PROGRAM PRG_08_AutoCrossCut
VAR
	iStep: INT;
	TON_DownDelay: TON;
	ctu_DoublePass: CTU;
	bDoublePassCountUp: BOOL;
	TON_bAutoUp: TON;
	bTON_AutoUp: BOOL;
	R_TRIG_0: R_TRIG;
	TON_AutoCrossCutError: TON;
	SR_DoublePass: SR;
	bDoublePassQ: BOOL;
	FB_Blinker_AutoCrossCut: fb_Blinker;
	TON_AutoCrossCutWatchdog: TON;
	RS_watchdog: RS;
	R_TRIG_1: R_TRIG;
	R_TRIG_2: R_TRIG;
	R_TRIG_3: R_TRIG;
	R_TRIG_4: R_TRIG;
	R_TRIG_5: R_TRIG;
	bWatchdogReset: BOOL;
	R_TRIG_6: R_TRIG;
	R_TRIG_7: R_TRIG;
	SR_WatchdogTriggered: SR;
	bWatchdogSet: BOOL;
	iStepErr: INT;
	R_TRIG_iStepErr: R_TRIG;
END_VAR

// Watchdog timeout error step
	R_TRIG_iStepErr(CLK:= SR_WatchdogTriggered.Q1, Q=> );
	IF R_TRIG_iStepErr.Q THEN
		iStepErr := iStep;
	ELSIF IN_FaultReset AND SR_WatchdogTriggered.Q1 THEN
		iStepErr := 0;
	END_IF

	
// error
	IF		NOT bSafetyOK 
			OR IN_FaultReset 
			OR NOT OUT_bSawON 
			OR bAnyServoError 
			OR bMachineHoming 
			OR bCrossCutPosition 
			OR SR_WatchdogTriggered.Q1
			OR bRemote
	THEN	iStep	:=	0 ;
			bWatchdogReset := TRUE ;
	END_IF

(* Time delay 0.5 sec after saw blade reached the bottom limit *)	
	TON_DownDelay(IN:= , PT:= T#0.5S, Q=> , ET=> );
	IF		iStep <> 30 THEN
			TON_DownDelay.IN	:= FALSE ;
	END_IF
(* Double Pass counter BOOL *)
	IF		ctu_DoublePass.CV	=	1
	THEN	bDoublePassCountUp		:=	TRUE;
	ELSE	bDoublePassCountUp		:=	FALSE;
	END_IF

CASE iStep OF 
	0:		//	Step 0	:	Init step
				bAutoCrossCut	:= FALSE ;
				bAutoUp			:= FALSE ;
				bAutoDown		:= FALSE ;
				bAutoCut		:= FALSE ;
				bAutoReturn		:= FALSE ;
				bTON_AutoUp		:= FALSE ;
				bWatchdogReset	:= TRUE  ;
				
		IF
				bSafetyOK
				AND bTurret045Range
				AND OUT_bSawON
				AND (bAutoCrossCutEnable AND IN_bAutoCycleStart AND NOT bRemote)
				AND NOT bMachineHoming
				AND NOT bCrossCutPosition
				AND bCarriageCentreRef
		THEN
				bAutoCrossCut := TRUE	;
				bWatchdogReset := TRUE  ;
				iStep	:=		20		;
		ELSE
				bAutoCrossCut := FALSE	;
				bWatchdogReset := FALSE ;
				iStep	:=		0		;
		END_IF

	20:		// Step 20	:	Saw RETURN movement
		IF 
				bAutoCrossCut
				AND bSafetyOK
				AND NOT bCrossCutRightLimit
			
		THEN	bAutoReturn	:=	TRUE	;
				bWatchdogReset := FALSE ;
		
		ELSE
				bAutoReturn	:=	FALSE	;
				bWatchdogReset := TRUE  ;
				iStep		:=	30		;
		END_IF
	
		IF 		NOT bSafetyOK
		THEN 	
				bAutoReturn	:=	FALSE	;
				bWatchdogReset := TRUE  ;
				iStep		:=	0		;
		END_IF
		
	30:		// Step 30	:	Saw DOWN movement
	ctu_DoublePass.CV;
		IF
				bAutoCrossCut
				AND bSafetyOK
				AND ((bAutoCrossCutDoublePass AND NOT bDoublePassReference AND bDoublePassCountUp) 
					OR ( NOT SR_DownLimit.Q1 AND (bDoublePassQ OR NOT bDoublePassCountUp)))
		THEN	
				bAutoDown	:=	TRUE	;
				bWatchdogReset := FALSE ;
		ELSE
				bAutoDown	:=	FALSE	;
				TON_DownDelay.IN := TRUE ;
					IF TON_DownDelay.Q THEN
						bWatchdogReset := TRUE ;
						iStep	:=	40		;
					END_IF
		END_IF
		
		IF 		NOT bSafetyOK
		THEN 	
				bAutoDown	:=	FALSE	;
				bWatchdogReset := TRUE  ;
				iStep		:=	0		;
		END_IF
	
	40:		// Step 40	:	Saw CUT movement
		IF
				bAutoCrossCut
				AND bSafetyOK
				AND	NOT bCrossCutLeftLimit
			THEN
				bAutoCut	:=	TRUE	;
				bWatchdogReset := FALSE ;
		ELSE
				bAutoCut	:=	FALSE	;
				bWatchdogReset := TRUE	;
				iStep		:=	50		;
		END_IF
		
		IF 		NOT bSafetyOK
			THEN 	
				bAutoCut	:=	FALSE	;
				bWatchdogReset := TRUE	;
				iStep		:=	0		;
		END_IF
	
	50:		// Step 50	:	Saw UP movement		(* for double pass: only lift slightly, RETURN, then plunge all the way down *)
	ctu_DoublePass.CV;	
		IF
				bAutoCrossCutDoublePass AND bDoublePassCountUp AND NOT bDoublePassQ
			THEN
				bTON_AutoUp	:=	TRUE	;
				bWatchdogReset := FALSE ;
				bAutoUp		:=	NOT TON_bAutoUp.Q	;
				
				IF
					R_TRIG_0.Q THEN
					bWatchdogReset := TRUE ;
					iStep	:=	60	;
				END_IF
				
		ELSIF
				bAutoCrossCut
				AND bSafetyOK
				AND NOT bSawUpLimit
				AND ((bDoublePassQ AND NOT bDoublePassCountUp AND bAutoCrossCutDoublePass) OR (NOT bAutoCrossCutDoublePass))
			THEN
				bAutoUp		:=	TRUE	;
				bWatchdogReset := FALSE ;
		ELSE
				bAutoUp		:=	FALSE	;
				bWatchdogReset := TRUE	;
				iStep		:=	60		;
		END_IF
		
		IF 		NOT bSafetyOK
		THEN 	
				bAutoUp		:=	FALSE	;
				bWatchdogReset := TRUE	;
				iStep		:=	0		;
		END_IF
	
	60:		// Step 60	:	Saw RETURN movement (loop back to step 20 if double pass)
		IF
				bAutoCrossCutDoublePass
				AND bDoublePassCountUp
		THEN
				bWatchdogReset := TRUE  ;
				iStep		:=	20		;
		ELSIF	
				bAutoCrossCut
				AND bSafetyOK
				AND NOT bCrossCutCentre
		THEN
				bWatchdogReset := FALSE ;
				bAutoReturn	:=	TRUE	;
		ELSE
				bAutoReturn	:=	FALSE	;
				bWatchdogReset := TRUE	;
				iStep		:=	0		;
		END_IF
		
		IF 		NOT bSafetyOK
		THEN 	
				bAutoReturn	:=	FALSE	;
				bWatchdogReset := TRUE	;
				iStep		:=	0		;
		END_IF
END_CASE

ACTION ACT_08_1_AutoCrossCut:
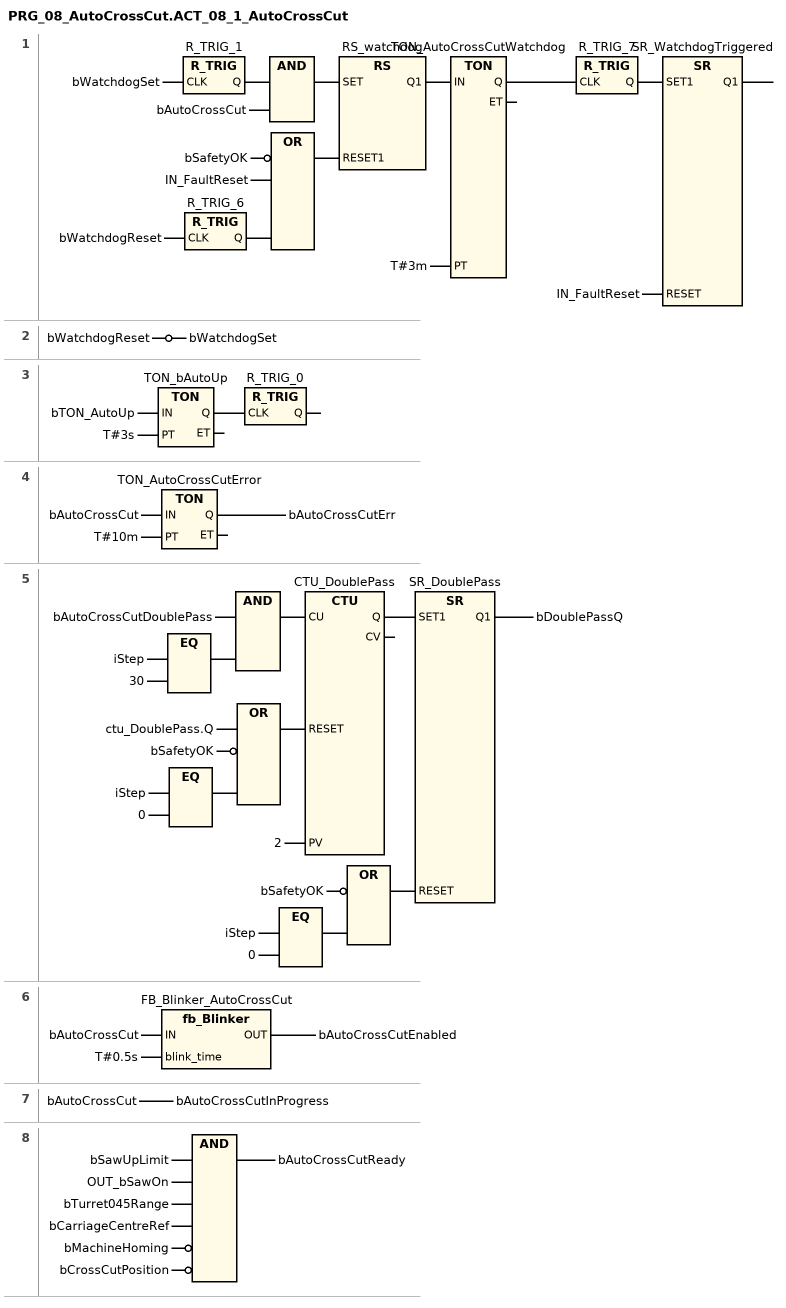
// NETWORK 1
R_TRIG_1(CLK := bWatchdogSet); // R_TRIG
R_TRIG_6(CLK := bWatchdogReset); // R_TRIG
RS_watchdog(SET := R_TRIG_1.Q AND bAutoCrossCut, RESET1 := NOT bSafetyOK OR IN_FaultReset OR R_TRIG_6.Q); // RS
TON_AutoCrossCutWatchdog(IN := RS_watchdog.Q1, PT := T#3m); // TON
R_TRIG_7(CLK := TON_AutoCrossCutWatchdog.Q); // R_TRIG
SR_WatchdogTriggered(SET1 := R_TRIG_7.Q, RESET := IN_FaultReset); // SR

// NETWORK 2
bWatchdogSet := NOT bWatchdogReset;

// NETWORK 3
TON_bAutoUp(IN := bTON_AutoUp, PT := T#3s); // TON
R_TRIG_0(CLK := TON_bAutoUp.Q); // R_TRIG

// NETWORK 4
TON_AutoCrossCutError(IN := bAutoCrossCut, PT := T#10m); // TON
bAutoCrossCutErr := TON_AutoCrossCutError.Q;

// NETWORK 5
CTU_DoublePass(
    CU := bAutoCrossCutDoublePass AND iStep = 30,
    RESET := ctu_DoublePass.Q OR NOT bSafetyOK OR iStep = 0,
    PV := 2); // CTU
SR_DoublePass(SET1 := CTU_DoublePass.Q, RESET := NOT bSafetyOK OR iStep = 0); // SR
bDoublePassQ := SR_DoublePass.Q1;

// NETWORK 6
FB_Blinker_AutoCrossCut(IN := bAutoCrossCut, blink_time := T#0.5s); // fb_Blinker
bAutoCrossCutEnabled := FB_Blinker_AutoCrossCut.OUT;

// NETWORK 7
bAutoCrossCutInProgress := bAutoCrossCut;

// NETWORK 8
bAutoCrossCutReady := bSawUpLimit AND OUT_bSawOn AND bTurret045Range AND bCarriageCentreRef AND NOT bMachineHoming AND NOT bCrossCutPosition;
END_ACTION

END_PROGRAM

(* stored: Version 1.1.0.1, ProductVersion 3.1.4024.15
   POU PRG_08_AutoCrossCut: Id {73f4070d-b53d-44b0-b7c0-d862c4fca4a8}, SpecialFunc None
   Action ACT_08_1_AutoCrossCut: Id {63a0db5e-5485-4feb-b0e7-b93f232749ba} *)
